{attribute 'qualified_only'}
{attribute 'strict'}
{attribute 'to_string'}
TYPE tyConveyorModeControl :
(
Standby 					:=0,
init 						:=10,
Stopped  					:=20,

//Cycle Steps 
WaitForBottle  				:=30,
OpenInfeedStopper  			:=40,
MoveToTestStation  			:=50,
ExtendTestHead  			:=60,
InjectAir  					:=70,
StabilizeAndMeasure  		:=80,
ReleaseTestHead  			:=90,
ReleaseBottle  				:=100,
RejectBottle  				:=110,

Fault  						:=999
);
END_TYPE

(* stored: Version 1.1.0.1
   DUT tyConveyorModeControl: Id {697a063f-445d-4c3c-aae2-d2265e720556} *)
